Universal Robots PolyScope program: realtime_control.urp

Program realtime_control (installation=default directory=/programs createdIn=5.24.0 lastSavedIn=5.24.0 robotSerialNumber=20215500838)
Calibrated DH parameters: a=[0.00019, -0.411898, -0.391136, 0.000062, -0.000012, 0]; d=[0.162688, -88.582522, 83.432095, 5.283837, 0.099747, 0.099603]; alpha=[1.571205, 0.001193, 0.006305, 1.569894, -1.57032, 0]; deltaTheta=[0, -0.251208, 6.451567, 0.082828, 0.000001, 0]
InitVariablesNode
Robot Program (runOnlyOnce=false)
  Loop Forever
    new_pos := p[read_input_float_register(0),read_input_float_register(1),read_input_float_register(2),read_input_float_register(3),read_input_float_register(4),read_input_float_register(5)]
    If new_pos != p[0,0,0,0,0,0]
      Script: servoj(get_inverse_kin(new_pos), t=0.5, lookahead_time=0.2, gain=100)
    Script: sync()
